TYPE ST_CoeEntry_DINT EXTENDS ST_CoeEntry :
STRUCT
	Value	: DINT;
END_STRUCT
END_TYPE

(* stored: Version 1.1.0.1, ProductVersion 3.1.4024.14
   DUT ST_CoeEntry_DINT: Id {16f6913e-13d1-080a-3b80-5da6f7cb44ad} *)
